// TIA Portal V19 export
ORGANIZATION_BLOCK "Main"   // OB2201, LAD, ProgramCycle
TITLE = "Main Program Sweep (Cycle)"
// stored: AutoNumber false, IsIECCheckEnabled true, Namespace Unit2.EM1, SetENOAutomatically true
   VAR_INPUT
      Initial_Call : Bool;   // Initial call of this OB
      Remanence : Bool;   // =True, if remanent data are available
   END_VAR
BEGIN

REGION Network 1 (SCL): Call Equipment
   "Unit2.EM1.instSimulation"();


   "Unit2.EM1.CallEquipment_DB"(unitStatus:="Unit2.EmNodes".unitStatus,
                    unitAlarmDB:="Unit2.Alarms".emAlarms[Unit2_EM1],
                    emFeedback:="Unit2.EmNodes".emFeedback[Unit2_EM1]);
END_REGION
END_ORGANIZATION_BLOCK
